FUNCTION F_GetDorPressure : real
VAR_INPUT
	nPressurePV:INT;
END_VAR

VAR
END_VAR

F_GetDorPressure := -190 * ((10 / 32767 ) * nPressurePV)+ 950;

END_FUNCTION

(* stored: Version 1.1.0.1, ProductVersion 3.1.4024.12
   POU F_GetDorPressure: Id {d5eb6636-a4af-417e-be51-f91c045e6ee3}, SpecialFunc None *)
